// TIA Portal V19 export
FUNCTION_BLOCK "MatCounter"   // FB123, LAD
TITLE = Material counter main
// stored: Access Published, MemoryReserve 100, SetENOAutomatically false
   VAR_INPUT
      CIn : "MatCountCIn";
      StandstillVelocityThreshold : LReal := 200.0;
      Config : Struct
         Default_FAK : LReal;
      END_STRUCT;
   END_VAR
   VAR_OUTPUT
      COut : Struct
         AlarmsPresence : Bool;
         WarningsPresence : Bool;
         StopFeeding : Bool;
         CounterValid : Bool;
         Standstill : Bool;
         PresetDone : Bool;
         ActualVelocity : LReal;
      END_STRUCT;
      Alr : Struct
         CounterNotInOperation : Bool;
      END_STRUCT;
      Wng : Struct
         EncoderNotValid : Bool;
         EncoderPosNotValid : Bool;
         PresetRunning : Bool;
      END_STRUCT;
   END_VAR
   VAR_IN_OUT
      PersistentValues : "MatCountPersistent";
   END_VAR
   VAR
      Status : Int;
      Sts : Struct
         PLCStartUpDone : Bool;
         Initialization : Bool;
         InOperation : Bool;
         PresetDone : Bool;
         FAKCalcDoneAndApply : Bool;
         RestorePreviousFAKDone : Bool;
         FAKManChangeApply : Bool;
         SetDefaultFAKDone : Bool;
         FAKManChange : Bool;
         HMIOperationDone : Bool;
         NewPositionToForce : LReal;
         NewFAK : LReal;
         VelocityLessThanThreshold : Bool;
      END_STRUCT;
      tonInOperation : TON_TIME;
      tonOpDone : TON_TIME;
      HMI : Struct
         PbFAKCalculation : Bool;
         PbFAKDefault : Bool;
         PbFAKPrevious : Bool;
         FAKSetDefaultDone : Bool;
         FAKCalcDone : Bool;
         FAKSetPrevDone : Bool;
         LenghtDesired : LReal;
         LenghtMeasured : LReal;
         FAKPrevious : LReal;
         FAKDefault : LReal;
      END_STRUCT;
      Aux : Struct
         PbFAKCalculation : Bool;
         PbFAKDefault : Bool;
         PbFAKPrevious : Bool;
      END_STRUCT;
      Check_Velocity { S7_SetPoint := 'True'} : "Check_Axis_Velocity";
   END_VAR
   VAR_TEMP
      InOperationCnd : Bool;
      ActualFAK : LReal;
      AxPosFAK : LReal;
      FAKCalculationExe : Bool;
      FAKDefaultExe : Bool;
      FAKPreviousExe : Bool;
   END_VAR
   VAR CONSTANT
      "0_INIT" : Int := 0;
      "1_IN_OPERATION" : Int := 1;
   END_VAR
   VAR_TEMP   // added for the SCL form of the ladder/FBD networks
      _w1 : Bool;
      _w2 : Bool;
      _w3 : Bool;
   END_VAR
BEGIN

REGION Network 1: Save persistent pos axis value
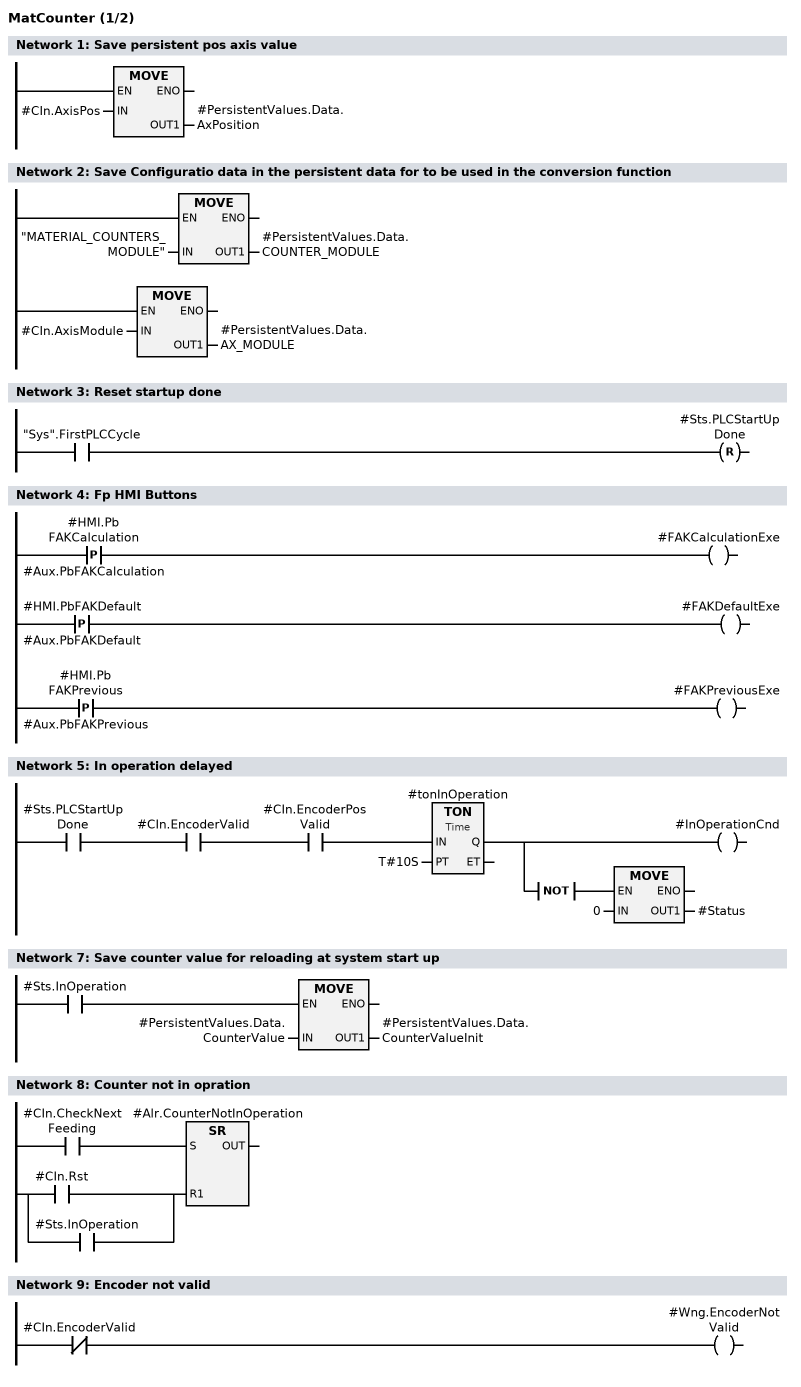
   RUNG wire#powerrail
      Move(in := #CIn.AxisPos, out1 => #PersistentValues.Data.AxPosition)
   END_RUNG
   // the same network as SCL:
   #PersistentValues.Data.AxPosition := #CIn.AxisPos;
END_REGION

REGION Network 2: Save Configuratio data in the persistent data for to be used in the conversion function
   RUNG wire#powerrail
      Move(in := "MATERIAL_COUNTERS_MODULE", out1 => #PersistentValues.Data.COUNTER_MODULE)
   END_RUNG
   RUNG wire#powerrail
      Move(in := #CIn.AxisModule, out1 => #PersistentValues.Data.AX_MODULE)
   END_RUNG
   // the same network as SCL:
   #PersistentValues.Data.COUNTER_MODULE := "MATERIAL_COUNTERS_MODULE";
   #PersistentValues.Data.AX_MODULE := #CIn.AxisModule;
END_REGION

REGION Network 3: Reset startup done
   RUNG wire#powerrail
      Contact( "Sys".FirstPLCCycle )
      R_Coil( #Sts.PLCStartUpDone )
   END_RUNG
   // the same network as SCL:
   IF "Sys".FirstPLCCycle THEN #Sts.PLCStartUpDone := FALSE; END_IF;
END_REGION

REGION Network 4: Fp HMI Buttons
   RUNG wire#powerrail
      P_Contact(operand := #HMI.PbFAKCalculation, bit := #Aux.PbFAKCalculation)
      Coil( #FAKCalculationExe )
   END_RUNG
   RUNG wire#powerrail
      P_Contact(operand := #HMI.PbFAKDefault, bit := #Aux.PbFAKDefault)
      Coil( #FAKDefaultExe )
   END_RUNG
   RUNG wire#powerrail
      P_Contact(operand := #HMI.PbFAKPrevious, bit := #Aux.PbFAKPrevious)
      Coil( #FAKPreviousExe )
   END_RUNG
   // the same network as SCL:
   #_w1 := #HMI.PbFAKCalculation AND NOT #Aux.PbFAKCalculation;   // rising edge of #HMI.PbFAKCalculation
   #Aux.PbFAKCalculation := #HMI.PbFAKCalculation;
   #FAKCalculationExe := #_w1;
   #_w2 := #HMI.PbFAKDefault AND NOT #Aux.PbFAKDefault;   // rising edge of #HMI.PbFAKDefault
   #Aux.PbFAKDefault := #HMI.PbFAKDefault;
   #FAKDefaultExe := #_w2;
   #_w3 := #HMI.PbFAKPrevious AND NOT #Aux.PbFAKPrevious;   // rising edge of #HMI.PbFAKPrevious
   #Aux.PbFAKPrevious := #HMI.PbFAKPrevious;
   #FAKPreviousExe := #_w3;
END_REGION

REGION Network 5: In operation delayed
   RUNG wire#powerrail
      Contact( #Sts.PLCStartUpDone )
      Contact( #CIn.EncoderValid )
      Contact( #CIn.EncoderPosValid )
      { S7_Templates := "time_type := Time" } #tonInOperation.TON(pt := T#10S, et =>)
      wire#w1
      Coil( #InOperationCnd )
   END_RUNG
   RUNG wire#w1
      Not()
      Move(in := 0, out1 => #Status)
   END_RUNG
   // the same network as SCL:
   #tonInOperation(IN := #Sts.PLCStartUpDone AND #CIn.EncoderValid AND #CIn.EncoderPosValid, PT := T#10S);   // TON
   #InOperationCnd := #tonInOperation.Q;
   IF NOT #tonInOperation.Q THEN #Status := 0; END_IF;
END_REGION

REGION Network 6 (SCL): Main
   CASE #Status OF

       #"0_INIT":

           //Reset several status
           #Sts.Initialization := TRUE;
           #Sts.InOperation := FALSE;
           #Sts.PresetDone := FALSE;
           #Sts.FAKCalcDoneAndApply := FALSE;
           #Sts.RestorePreviousFAKDone := FALSE;
           #Sts.FAKManChangeApply := FALSE;



           // Check FAK Value
           IF (#PersistentValues.Data.FAK < "FAK_MIN_VALUE") OR (#PersistentValues.Data.FAK > "FAK_MAX_VALUE") THEN
               #PersistentValues.Data.FAK := #Config.Default_FAK;
           END_IF;

           #PersistentValues.Data.FAK := #PersistentValues.Par.FAK;

           //If conditions are ok then start
           IF #InOperationCnd THEN

               IF #PersistentValues.Data.CounterValueInit > 0.0 THEN
                   #Sts.NewPositionToForce := #PersistentValues.Data.CounterValueInit;
               ELSE
                   #Sts.NewPositionToForce := 0.0;
               END_IF;

               #AxPosFAK := #PersistentValues.Data.AxPosition * #PersistentValues.Data.FAK;
               #PersistentValues.Data.CounterOffset := #Sts.NewPositionToForce - #AxPosFAK;

               //Update counter
               "MatCounter_UPD"(Data := #PersistentValues.Data);

               #Status := #"1_IN_OPERATION";
           END_IF;

       #"1_IN_OPERATION":

           #Sts.Initialization := FALSE;
           #Sts.InOperation := TRUE;

           //Update counter
           "MatCounter_UPD"(Data:=#PersistentValues.Data);


           //=====================================================
           //PRESET
           //=====================================================
           IF #CIn.PresetExe AND NOT #Sts.PresetDone THEN
               #Sts.NewPositionToForce := #CIn.PresetPosition;
               #AxPosFAK := #PersistentValues.Data.AxPosition * #PersistentValues.Data.FAK;
               #PersistentValues.Data.CounterOffset := #Sts.NewPositionToForce - #AxPosFAK;

               //Update counter
               "MatCounter_UPD"(Data := #PersistentValues.Data);

               #Sts.PresetDone := TRUE;
           END_IF;

           IF NOT #CIn.PresetExe AND #Sts.PresetDone THEN
               #Sts.PresetDone := FALSE;
           END_IF;

           //=====================================================
           //NEW FAK
           //=====================================================
           IF #FAKCalculationExe AND NOT #Sts.FAKCalcDoneAndApply THEN

               #Sts.NewPositionToForce := #PersistentValues.Data.CounterValue;

               #Sts.NewFAK := ( #HMI.LenghtMeasured / #HMI.LenghtDesired ) * #PersistentValues.Data.FAK;

               #PersistentValues.Data.FAKPrevious := #PersistentValues.Data.FAK;
               #PersistentValues.Data.FAK := #Sts.NewFAK;
               #PersistentValues.Par.FAK := #Sts.NewFAK;
               #HMI.LenghtMeasured := #HMI.LenghtDesired;

               #AxPosFAK := #PersistentValues.Data.AxPosition * #PersistentValues.Data.FAK;
               #PersistentValues.Data.CounterOffset := #Sts.NewPositionToForce - #AxPosFAK;

               //Update counter
               "MatCounter_UPD"(Data := #PersistentValues.Data);

               #Sts.FAKCalcDoneAndApply := TRUE;
           END_IF;
           //=====================================================
           //DEFAULT FAK
           //=====================================================
           IF #FAKDefaultExe AND NOT #Sts.SetDefaultFAKDone THEN
               #Sts.NewPositionToForce := #PersistentValues.Data.CounterValue;
               #Sts.NewFAK := #Config.Default_FAK;
               #PersistentValues.Data.FAKPrevious := #PersistentValues.Data.FAK;
               #PersistentValues.Data.FAK := #Sts.NewFAK;
               #PersistentValues.Par.FAK := #Sts.NewFAK;
               #AxPosFAK := #PersistentValues.Data.AxPosition * #PersistentValues.Data.FAK;
               #PersistentValues.Data.CounterOffset := #Sts.NewPositionToForce - #AxPosFAK;

               //Update counter
               "MatCounter_UPD"(Data := #PersistentValues.Data);

               #Sts.SetDefaultFAKDone := TRUE;
           END_IF;
           //=====================================================
           //PREVIOUS FAK
           //=====================================================
           IF #FAKPreviousExe AND NOT #Sts.FAKCalcDoneAndApply THEN
               #Sts.NewPositionToForce := #PersistentValues.Data.CounterValue;
               #Sts.NewFAK := #PersistentValues.Data.FAKPrevious;
               #PersistentValues.Data.FAKPrevious := #PersistentValues.Data.FAK;
               #PersistentValues.Data.FAK := #Sts.NewFAK;
               #PersistentValues.Par.FAK := #Sts.NewFAK;
               #AxPosFAK := #PersistentValues.Data.AxPosition * #PersistentValues.Data.FAK;
               #PersistentValues.Data.CounterOffset := #Sts.NewPositionToForce - #AxPosFAK;
               //Update counter
               "MatCounter_UPD"(Data := #PersistentValues.Data);

               #Sts.RestorePreviousFAKDone := TRUE;
           END_IF;
           //=====================================================
           //MANUAL FAK
           //=====================================================
           IF #Sts.FAKManChange AND NOT #Sts.FAKManChangeApply THEN
               #Sts.NewPositionToForce := #PersistentValues.Data.CounterValue;
               #Sts.NewFAK := #PersistentValues.Par.FAK;
               #PersistentValues.Data.FAKPrevious := #PersistentValues.Data.FAK;
               #PersistentValues.Data.FAK := #Sts.NewFAK;
               #PersistentValues.Par.FAK := #Sts.NewFAK;
               #AxPosFAK := #PersistentValues.Data.AxPosition * #PersistentValues.Data.FAK;
               #PersistentValues.Data.CounterOffset := #Sts.NewPositionToForce - #AxPosFAK;

               //Update counter
               "MatCounter_UPD"(Data := #PersistentValues.Data);

               #Sts.FAKManChangeApply := TRUE;
           END_IF;
   END_CASE;
END_REGION

REGION Network 7: Save counter value for reloading at system start up
   RUNG wire#powerrail
      Contact( #Sts.InOperation )
      Move(in := #PersistentValues.Data.CounterValue, out1 => #PersistentValues.Data.CounterValueInit)
   END_RUNG
   // the same network as SCL:
   IF #Sts.InOperation THEN
       #PersistentValues.Data.CounterValueInit := #PersistentValues.Data.CounterValue;
   END_IF;
END_REGION

REGION Network 8: Counter not in opration
   RUNG wire#powerrail
      Contact( #CIn.CheckNextFeeding )
      S_SR(operand := #Alr.CounterNotInOperation, r1 := wire#w1)
   END_RUNG
   RUNG wire#powerrail
      Contact( #CIn.Rst )
   END_RUNG wire#w1
   RUNG wire#powerrail
      Contact( #Sts.InOperation )
   END_RUNG wire#w1
   // the same network as SCL:
   IF #CIn.CheckNextFeeding THEN
       #Alr.CounterNotInOperation := TRUE;   // SR flip-flop
   END_IF;
   IF #CIn.Rst OR #Sts.InOperation THEN #Alr.CounterNotInOperation := FALSE; END_IF;
END_REGION

REGION Network 9: Encoder not valid
   RUNG wire#powerrail
      I_Contact( #CIn.EncoderValid )
      Coil( #Wng.EncoderNotValid )
   END_RUNG
   // the same network as SCL:
   #Wng.EncoderNotValid := NOT #CIn.EncoderValid;
END_REGION

REGION Network 10: Encoder pos not valid
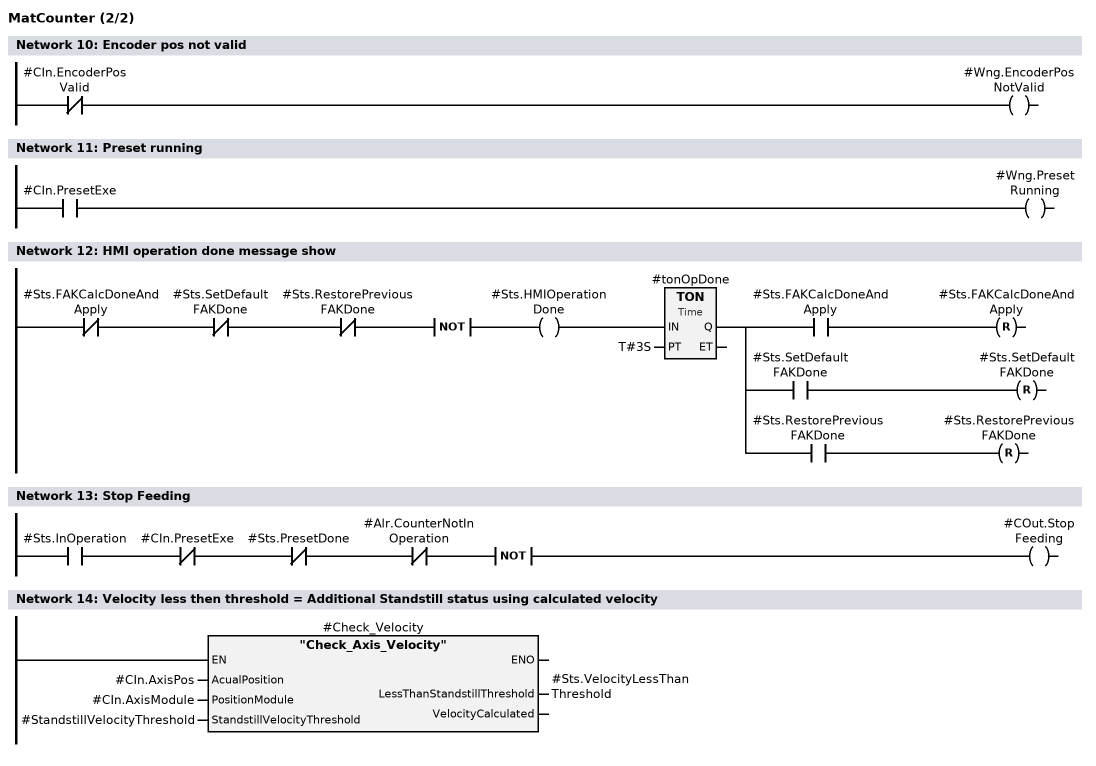
   RUNG wire#powerrail
      I_Contact( #CIn.EncoderPosValid )
      Coil( #Wng.EncoderPosNotValid )
   END_RUNG
   // the same network as SCL:
   #Wng.EncoderPosNotValid := NOT #CIn.EncoderPosValid;
END_REGION

REGION Network 11: Preset running
   RUNG wire#powerrail
      Contact( #CIn.PresetExe )
      Coil( #Wng.PresetRunning )
   END_RUNG
   // the same network as SCL:
   #Wng.PresetRunning := #CIn.PresetExe;
END_REGION

REGION Network 12: HMI operation done message show
   RUNG wire#powerrail
      I_Contact( #Sts.FAKCalcDoneAndApply )
      I_Contact( #Sts.SetDefaultFAKDone )
      I_Contact( #Sts.RestorePreviousFAKDone )
      Not()
      Coil( #Sts.HMIOperationDone )
      { S7_Templates := "time_type := Time" } #tonOpDone.TON(pt := T#3S, et =>)
      wire#w1
      Contact( #Sts.FAKCalcDoneAndApply )
      R_Coil( #Sts.FAKCalcDoneAndApply )
   END_RUNG
   RUNG wire#w1
      Contact( #Sts.SetDefaultFAKDone )
      R_Coil( #Sts.SetDefaultFAKDone )
   END_RUNG
   RUNG wire#w1
      Contact( #Sts.RestorePreviousFAKDone )
      R_Coil( #Sts.RestorePreviousFAKDone )
   END_RUNG
   // the same network as SCL:
   #Sts.HMIOperationDone := NOT (NOT #Sts.FAKCalcDoneAndApply AND NOT #Sts.SetDefaultFAKDone AND NOT #Sts.RestorePreviousFAKDone);
   #tonOpDone(IN := #Sts.HMIOperationDone, PT := T#3S);   // TON
   IF #tonOpDone.Q AND #Sts.FAKCalcDoneAndApply THEN #Sts.FAKCalcDoneAndApply := FALSE; END_IF;
   IF #tonOpDone.Q AND #Sts.SetDefaultFAKDone THEN #Sts.SetDefaultFAKDone := FALSE; END_IF;
   IF #tonOpDone.Q AND #Sts.RestorePreviousFAKDone THEN #Sts.RestorePreviousFAKDone := FALSE; END_IF;
END_REGION

REGION Network 13: Stop Feeding
   RUNG wire#powerrail
      Contact( #Sts.InOperation )
      I_Contact( #CIn.PresetExe )
      I_Contact( #Sts.PresetDone )
      I_Contact( #Alr.CounterNotInOperation )
      Not()
      Coil( #COut.StopFeeding )
   END_RUNG
   // the same network as SCL:
   #COut.StopFeeding := NOT (#Sts.InOperation AND NOT #CIn.PresetExe AND NOT #Sts.PresetDone AND NOT #Alr.CounterNotInOperation);
END_REGION

REGION Network 14: Velocity less then threshold = Additional Standstill status using calculated velocity
   RUNG wire#powerrail
      #Check_Velocity(AcualPosition := #CIn.AxisPos, PositionModule := #CIn.AxisModule, StandstillVelocityThreshold := #StandstillVelocityThreshold, LessThanStandstillThreshold => #Sts.VelocityLessThanThreshold, VelocityCalculated =>)
   END_RUNG
   // the same network as SCL:
   #Check_Velocity(AcualPosition := #CIn.AxisPos,   // "Check_Axis_Velocity"
                   PositionModule := #CIn.AxisModule,
                   StandstillVelocityThreshold := #StandstillVelocityThreshold,
                   LessThanStandstillThreshold => #Sts.VelocityLessThanThreshold);
END_REGION

REGION Network 15 (SCL): Update status
   #COut.AlarmsPresence := #Alr.CounterNotInOperation;
   #COut.WarningsPresence := #Wng.EncoderNotValid OR #Wng.EncoderPosNotValid OR #Wng.PresetRunning;
   #COut.CounterValid := #Sts.InOperation;
   #COut.Standstill := #CIn.Standstill AND #Sts.VelocityLessThanThreshold;
   #COut.PresetDone := #Sts.PresetDone;

   #COut.ActualVelocity := #Check_Velocity.VelocityCalculated;


   #PersistentValues.Data.CounterValid := #COut.CounterValid;
   #PersistentValues.Data.Standstill := #COut.Standstill;
END_REGION

REGION Network 16 (SCL): HMI
   IF NOT #Sts.PLCStartUpDone THEN
       #PersistentValues.Par.FAK := #PersistentValues.Data.FAK;
       #HMI.PbFAKCalculation := FALSE;
       #HMI.PbFAKDefault := FALSE;
       #HMI.PbFAKPrevious := FALSE;
       #Sts.PLCStartUpDone := TRUE;
   END_IF;

   //Check FAK Value
   #PersistentValues.Par.FAK := LIMIT_LREAL(IN := #PersistentValues.Par.FAK, MN := "FAK_MIN_VALUE", MX := "FAK_MAX_VALUE");





   //HMI Change value
   #Sts.FAKManChange := #PersistentValues.Par.FAK <> #PersistentValues.Data.FAK;

   IF NOT #Sts.FAKManChange THEN
       #Sts.FAKManChangeApply := FALSE;
   END_IF;

   #HMI.FAKDefault := #Config.Default_FAK;
   #HMI.FAKPrevious := #PersistentValues.Data.FAKPrevious;

   #HMI.FAKSetDefaultDone := #Sts.HMIOperationDone AND #Sts.SetDefaultFAKDone;
   #HMI.FAKCalcDone := #Sts.HMIOperationDone AND #Sts.FAKCalcDoneAndApply;
   #HMI.FAKSetPrevDone := #Sts.HMIOperationDone AND #Sts.RestorePreviousFAKDone;
END_REGION
END_FUNCTION_BLOCK
